# B&R Automation Studio project dbserv_0640 (part 2)

### dbvist.h
```c
/************************************************************************/
/*	Headerfile für DbVist												*/
/*																		*/
/************************************************************************/
#include "pwi_lib.h"

/* Tasknamen für Versionsanzeige */
#define	TASK_DBSERV		"dbserv"
#define	TASK_DBSTCP		"dbstcp"
#define	TASK_DBVIST		"dbvist"
#define	TASK_IEC103		"iec103"
#define	TASK_L2DP		"l2dp"
#define	TASK_IODRV		"iodrv"
#define	TASK_GPS		"gps"

#define	MAX_ITEM			4000	/* max.Anzahl von Items */
#define ANZ_SCAN_AL			64		/* gescannte Alarme pro Zyklus */

#define	MENU_MAIN	1
#define	MENU_ITEM	2
#define	MENU_ALISTE	3
#define	MENU_NODP	5
#define	MENU_SYS	6
#define	MENU_CLOCK	7
#define	MENU_VERSION	8
#define MENU_MAX	10

#define KEY_OPT		33
#define KEY_F		34
#define KEY_STERN	35
#define KEY_ALISTE	39
#define KEY_AP		40
#define KEY_BP		41
#define KEY_AL		42
#define KEY_ZL		43
#define KEY_Q		48
#define KEY_SYS		51
#define KEY_PAGEUP	53
#define KEY_ONEUP	54
#define KEY_PLUS	55
#define KEY_PAGEDWN	56
#define KEY_ONEDWN	57
#define KEY_MINUS	58
#define KEY_UP		59
#define KEY_RIGHT	60
#define KEY_DOWN	61
#define KEY_LEFT	62
#define KEY_HOME	63
#define KEY_ENTER	65

typedef struct {
	STRING	time[32];
} ALTIME_typ;

/*
typedef struct {
	UINT	LifeCheck;
	UINT	TimeOut;
	INT		DefcurNo;
	INT		DefcmdNo;
	INT		NewcurNo;
	INT		NewcmdNo;
	USINT	DefownPage;
	USINT	NewownPage;
	SINT	DefcurPage;
	SINT	NewcurPage;
	USINT	triggerCur;
	USINT	disCursor;
	USINT	disCurLFRG;
	SINT	nextInpENo;
	SINT	nextInpESt;
	USINT	loopInput;
	USINT	disInput;
	USINT	disKey;
	USINT	signKey;
	USINT	dpChar;
	USINT	dpFix;
	USINT	hiddenChar;
	USINT	strInsert;
	USINT	srcKeyLim;
	USINT	curChar;
	USINT	curInput;
	SINT	curPosObj;
	USINT	signFormat;
	USINT	optNewPage;
	USINT	nNCnewPage;
	USINT	nNXnewPage;
	USINT	notValidChar;
} PWI_env;
*/
typedef struct {
	UINT	PwiStep;
	BOOL	okPWI;
	UDINT	idPWI;
	UINT	codePWI;
	UINT	infoPWINo;
	UINT	infoPWILn;
	UINT	waitCycles;
	UINT	stateOut;
	USINT	szTrends[256];
	USINT	SpeechEnab[256];
	UINT	SpeechAct;
	UINT	PageAct;
	BOOL	PageAgain;
	BOOL	PageReady;
	UINT	PageNew;
	UINT	SpeechNew;
	INT		ActcurNo;
	INT		ActcmdNo;
	INT		ActownPage;
	USINT	KeyFieldT[16];
	USINT	KeyField[16];
	USINT	KeyFieldP[16];
	USINT	KeyFieldO[16];
	BOOL	TableauOK;
	BOOL	keypress;
	BOOL	keypuls;
	USINT	keyold;
	USINT	keycode;
	USINT	keycodeTab;
	USINT	messageTab;
	BOOL	enterpuls;
	UINT	stateCanTX;
	UINT	stateCanRX;
	UDINT	idCAN;
	UINT	nodeCAN;
	UINT	errCAN;
	USINT	Device[32];
	UINT	stateRsTX;
	UINT	stateRsRX;
	UDINT	idRS;
	UINT	argc;
	UDINT	argv[32];
	USINT	keyuser;
	USINT	ASCIIuser;
	BOOL	changePuls;
	BOOL	changepuls;
	BOOL	inputopen;
	BOOL	funcInp;
	USINT	funcEnter;
	BOOL	funcInpRun;
	UINT	stateInp;

	UINT	codePwi;
	UINT	infoPwi1;
	UINT	infoPwi2;

	UINT	codeText;
	UINT	infoTextNo;
	UINT	infoTextLn;

	UINT	codeMask;
	UINT	infoMaskNo;
	UINT	infoMaskLn;

	UINT	codePage;
	UINT	infoPageNo;
	UINT	infoPageLn;

	UINT	codeObj;
	UINT	infoObjNo;
	UINT	infoObjLn;

	UINT	codeGrph;
	UINT	infoGrphNo;
	UINT	infoGrphLn;

	UINT	codeTrend;
	UINT	infoTrendNo;
	UINT	infoTrendLn;

	UINT	codeCan;
	UDINT	infoCan1;
	UDINT	infoCan2;

	UINT	codeRs;
	UDINT	infoRs1;
	UDINT	infoRs2;

	PWI_env	envPWI;
} PWI_INTERFACE;

typedef struct {
	STRING	vers_dbserv[40];
	STRING	vers_dbvist[40];
	STRING	vers_dbstcp[40];
	STRING	vers_iec103[40];
	STRING	vers_l2dp[40];
	STRING	vers_iodrv[40];
	STRING	vers_gps[40];
} VERSION_typ;

/*_GLOBAL	UINT	PageAct,PageNew,,SpeechAct,SpeechNew;
_GLOBAL	BOOL	keypuls,;
_GLOBAL	USINT	keycode;
*/
_LOCAL	PWI_INTERFACE	*pPWI_INTERFACE;
_LOCAL	UDINT	lenPWI_INTERFACE;
_LOCAL	UINT	PageLast;
_LOCAL	BOOL	keypuls_old;

_LOCAL	STRING	UstName[32],Filter[32],FilterUnten[41];
_LOCAL	USINT	enableItem[MAX_ITEM];
_LOCAL	INT		UstNr;

_LOCAL	UINT	testUINT;
_LOCAL	UINT	GrpIdx,DTypIdx,DPIdx;
_LOCAL	USINT	enableGrp,enableDT,enableDP,enableOGrp,enableODT,enableODP;
_LOCAL	USINT	enableGrp_old,enableDT_old,indexGrp_old,indexDT_old;
_LOCAL	BOOL	activGrp,activDT,activDP;
_LOCAL	BOOL	activGrp_old,activDT_old;
_LOCAL	BOOL	setClock,enableSet,activSet,setClockStarted;
_LOCAL	RTCtime_typ	RTCtime,RTCtimeSet;
_LOCAL	INT		indexSYS, indexGrp,indexDT,indexDP,indexItem,indexAP,indexBP,indexAL,indexZL,indexALL;
_LOCAL	USINT	minute_old;
_LOCAL	UINT	AnzDPfiltered,LastFiltered;

_LOCAL void (*pInitPic[MENU_MAX])();
_LOCAL void (*pCyclPic[MENU_MAX])();
_LOCAL void (*pKeysPic[MENU_MAX])();

_LOCAL	UDINT	myidBrServer;
_LOCAL	UINT	statePV_xgetadr,CheckPWIerrors	_VAR_RETAIN;
_LOCAL 	UINT	idstat,brstate;
_LOCAL	UINT	scanAL,countAL,aktiveAlarme,countALGRP[MAX_GRP],aktiveAlarmeGrp[MAX_GRP];
_LOCAL	BOOL	SammStoer,GrpStoer[MAX_GRP];
_LOCAL	USINT	LED_Aliste;
_LOCAL	USINT	*pData_extern, *pData_iextern, *pData_intern, *pData_valid, *pData_time, *pData_itime, *pData_writelink, *pData_ieventlink, *pData_ihyst, *pData_ievent;
_LOCAL	UDINT 	length_extern, length_intern, length_iextern, length_valid, length_time, length_itime, length_writelink, length_ieventlink, length_ihyst, length_ievent;
_LOCAL	UINT	infoerror,LatchStatusSetValueItem;
_LOCAL	BOOL	Quitt;
_LOCAL	UINT	quitIndex;
_LOCAL	VERSION_typ	Version;
_LOCAL MoVerStruc_typ MO_ver_struct;
_LOCAL	STRING	TestText1[256],TestText2[256];
_LOCAL	UINT	TestTextNr;
```

### dbv_parse.h
```c
/******************************************************************************
*  Projekt:  DbVist Visualisierung für DbServ
*  Teil:     Parserfunktionen
*  Datei:    dbv_parse.c
*------------------------------------------------------------------------------
*  Revision: 01.00
*  Datum:    04-0-2006
*  Autor:    WAI
*------------------------------------------------------------------------------
*  Funktion:
*------------------------------------------------------------------------------
*  Rev.  | Datum    | Name | Kommentar
*  ------+----------+------+---------------------------------------------------
*  01.00 | 04-06-06 | WAI  | Datei-Erstellung
*        |          |      |
******************************************************************************/
/***********************************************************************/
/* Konstantendefinition                                                */
/***********************************************************************/
#define ERR_MSG_PRE_STRG				"dbv"
#define MAX_ERROR_MSG_LOG				20				/* Anzahl Fehler, die in das Log-Buch eingetragen werden */
/* Bezeichnung der Datenmodule */
#define DATA_OBJEKT_DPLIST		"dplist"
#define DATA_OBJEKT_TYPLIST		"typlist"
#define DATA_OBJEKT_DBVTEXT 	"dbv_text"
#define DATA_OBJEKT_TEXT1 		"text_1"
#define DATA_OBJEKT_TEXT2 		"text_2"
#define DATA_OBJEKT_PAGE 		"page_1"
#define DATA_OBJEKT_OBJ1 		"obj_1"
#define DATA_OBJEKT_OBJ2 		"obj_2"
#define DATA_OBJEKT_OBJ3 		"obj_3"
#define DATA_OBJEKT_OBJ4 		"obj_4"
#define DATA_OBJEKT_OBJ5 		"obj_5"

/* Delimiter */
#define DELIM_ALLGEMEIN_ANF		"<Allgemein>"
#define DELIM_ALLGEMEIN_END		"</Allgemein>"
#define DELIM_DTYP_ANF			"<Dtyp>"
#define DELIM_DTYP_END			"</Dtyp>"
#define DELIM_OBJGRPDTYP_ANF	"<ObjGrpDtyp>"
#define DELIM_OBJGRPDTYP_END	"</ObjGrpDtyp>"
#define DELIM_OBJITEMAP_ANF		"<ObjItemAP>"
#define DELIM_OBJITEMAP_END		"</ObjItemAP>"
#define DELIM_OBJITEMBPAL_ANF	"<ObjItemBPAL>"
#define DELIM_OBJITEMBPAL_END	"</ObjItemBPAL>"
#define DELIM_OBJITEMZL_ANF		"<ObjItemZL>"
#define DELIM_OBJITEMZL_END		"</ObjItemZL>"
#define DELIM_OBJITEMALIST_ANF	"<ObjItemAList>"
#define DELIM_OBJITEMALIST_END	"</ObjItemAList>"
#define DELIM_OBJSYS_ANF		"<ObjSys>"
#define DELIM_OBJSYS_END		"</ObjSys>"
#define DELIM_PAGE_ANF 			"<Page>"
#define DELIM_PAGE_END 			"</Page>"

/* Skalierungsparameter */
#define	MAX_DT					10		/* max.Anzahl von Datentypen */
#define	MAX_GRP					100		/* max.Anzahl von Gruppen */
#define	MAX_UNIT				32		/* max.Anzahl von Einheiten */
#define	MAX_TEXTLIST			32		/* max.Anzahl von Textlisten */
#define	MAX_TEXTVALUE			16		/* max.Wert einer Textliste */

#define BOOL_TYP						"_BOOL"
#define BOOL_IDX						0
#define USINT_TYP						"_USINT"
#define USINT_IDX						1
#define SINT_TYP						"_SINT"
#define SINT_IDX						2
#define UINT_TYP						"_UINT"
#define UINT_IDX						3
#define INT_TYP							"_INT"
#define INT_IDX							4
#define UDINT_TYP						"_UDINT"
#define UDINT_IDX						5
#define DINT_TYP						"_DINT"
#define DINT_IDX						6
#define REAL_TYP						"_REAL"
#define REAL_IDX						8
#define DOUBLE_TYP						"_DOUBLE"
#define DOUBLE_IDX						9

#define DTYP_AP							1
#define DTYP_BP							2
#define DTYP_AL							3
#define DTYP_ZL							4

/*-------------------------------------------------------
	Fehlermeldungen
---------------------------------------------------------*/
#define NO_ERROR						0

/* Fehlermeldungen: Datenmodul nicht gefunden */
#define PARS_ERR_DPLIST_NOT_FOUND		501				/* Fehler: Datenmodul dplist nicht gefunden */
#define PARS_TXT_DPLIST_NOT_FOUND		"datamodule dplist not found"

#define PARS_ERR_TYPLIST_NOT_FOUND		502				/* Fehler: Datenmodul typlist nicht gefunden */
#define PARS_TXT_TYPLIST_NOT_FOUND		"datamodule typlist not found"

#define PARS_ERR_DBVTEXT_NOT_FOUND		503				/* Fehler: Datenmodul dbv_text nicht gefunden */
#define PARS_TXT_DBVTEXT_NOT_FOUND		"datamodule dbv_text not found"

#define PARS_ERR_MEM_ALLOC				504				/* Fehler: Speicher kann nicht allokiert werden */
#define PARS_TXT_MEM_ALLOC				"TMP_alloc not successfull"

#define PARS_ERR_CREATE_DM				505				/* Fehler: Datenmodul kann nicht erzeugt werden */
#define PARS_TXT_CREATE_DM				"Create DM not successfull"

/* Fehlermeldungen des globalen Teiles */
#define PARS_ERR_UNKNOWN_GLOBAL_ENTRY	505				/* Fehler: Unbekannter Eintrag in globalen Bereich */
#define PARS_ERR_GRP_UNKNOWN			506				/* Fehler: Name kann keiner Gruppe zugeordnet werden */
#define PARS_ERR_TO_MUCH_GRP			507				/* Fehler: Anzahl deklarierter Gruppen zu gross  */
#define PARS_ERR_UNIT_UNKNOWN			508				/* Fehler: Name kann keiner Einheit zugeordnet werden */
#define PARS_ERR_TO_MUCH_UNITS			509				/* Fehler: Anzahl deklarierter Einheiten zu gross  */
#define PARS_ERR_TLIST_UNKNOWN			510				/* Fehler: Name kann keiner Textliste zugeordnet werden */
#define PARS_ERR_TO_MUCH_TLISTS			511				/* Fehler: Anzahl deklarierter Textlisten zu gross  */

#define PARS_ERR_DPTYP_NR_NOT_DEFINED	609				/* Fehler: Datentyp Nummer nicht definiert */
#define PARS_ERR_ITEM_NR_NOT_DEFINED	610				/* Fehler: Item Nummer nicht definiert */
#define PARS_ERR_ITEM_TYP_NOT_DEFINED	611				/* Fehler: Item Typ nicht definiert */
#define PARS_ERR_ITEM_TYP_UNKNOWN		612				/* Fehler: Item Typ unbekannt */
#define PARS_ERR_ITEM_NAME_NOT_DEFINED	613				/* Fehler: Item Name nicht definiert */

/* Fehlermeldungen des Itembereiches */
#define PARS_ERR_UNKNOWN_ITEM_ENTRY		700				/* Fehler: Unbekannter Eintrag in Item Bereich (DM typlist)*/
#define PARS_ERR_GRP_NOTDEFINED			701				/* Fehler: Gruppe ist nicht definiert */
#define PARS_ERR_TLIST_NOTDEFINED		702				/* Fehler: Textliste ist nicht definiert */
#define PARS_ERR_ITEM_DTYP_NOT_DEFINED	703				/* Fehler: Datentyp ist nicht definiert */

#define PARS_ERR_REPLACE				710				/* Fehler beim ersetzen von Token */

#define PARS_ERR_PWI_NOT_FOUND			800				/* Fehler: Interface zu PWI nicht gefunden */
#define PARS_ERR_PWI_ERROR				801				/* Fehler: PWI meldet Fehler */
/*-------------------------------------------------------
	Schlüsselworte
---------------------------------------------------------*/
/* Hilfskonstanten */

#define ALL_SECTION						0				/* Es wird im allgemeinen Teil geparst (Meldungsunterdrückung) */
#define DBV_SECTION						1				/* Es wird im VIS - Teil geparst (Meldung bei unbekannten Schlüsselworten) */
#define DP_PART							0				/* Es wird im allgemeinen Datenpunktbereich geparst */
#define ITEM_PART						1				/* Es wird im allgemeinen Itembereich geparst */

/* Schluesselworte Sectionen */
#define	KW_DBV_SECTION					"VIS"			/* Schlüsselwort für VIS-Section */
#define	KW_ALL_SECTION					"ALL"			/* Schlüsselwort für Allgemeine-Section */
#define KW_ITEM_SECTION					"ITEM"			/* Schlüsselwort für ITEM-Section */
#define KW_BLOCK_SECTION				"BLOCK"			/* Schlüsswlwort für Blockdefinition */

/* Schluesselworte  globaler Teil */
#define KW_UST							"UST"			/* Schlüsselwort für UST */
#define KW_VIS_USTNR					"NR"			/* Schlüsselwort für UST-Nummer */
#define KW_VIS_USTNAME					"NAME"			/* Schlüsselwort für UST-Name */
#define KW_VIS_USTIF					"IF"			/* Schlüsselwort für Interface */
#define KW_VIS_GRP						"GRP"			/* Schlüsselwort für Gruppe */
#define KW_VIS_GRPNAME					"NAME"			/* Schlüsselwort für Gruppennamen */
#define KW_VIS_UNIT						"EINH"			/* Schlüsselwort für Einheit */
#define KW_VIS_TLIST					"TLIST"			/* Schlüsselwort für Textliste */
#define KW_VIS_TLISTT0					"T0"			/* Schlüsselwort für Textliste Zusatnd 0*/
#define KW_VIS_TLISTT1					"T1"			/* Schlüsselwort für Textliste Zusatnd 1*/
#define KW_VIS_TLISTT2					"T2"			/* Schlüsselwort für Textliste Zusatnd 2*/
#define KW_VIS_TLISTT3					"T3"			/* Schlüsselwort für Textliste Zusatnd 3*/
#define KW_VIS_TLISTT4					"T4"			/* Schlüsselwort für Textliste Zusatnd 4*/
#define KW_VIS_TLISTT5					"T5"			/* Schlüsselwort für Textliste Zusatnd 5*/
#define KW_VIS_TLISTT6					"T6"			/* Schlüsselwort für Textliste Zusatnd 6*/
#define KW_VIS_TLISTT7					"T7"			/* Schlüsselwort für Textliste Zusatnd 7*/
#define KW_VIS_TLISTT8					"T8"			/* Schlüsselwort für Textliste Zusatnd 8*/
#define KW_VIS_TLISTT9					"T9"			/* Schlüsselwort für Textliste Zusatnd 9*/
#define KW_VIS_TLISTT10					"T10"			/* Schlüsselwort für Textliste Zusatnd 10*/
#define KW_VIS_TLISTT11					"T11"			/* Schlüsselwort für Textliste Zusatnd 11*/
#define KW_VIS_TLISTT12					"T12"			/* Schlüsselwort für Textliste Zusatnd 12*/
#define KW_VIS_TLISTT13					"T13"			/* Schlüsselwort für Textliste Zusatnd 13*/
#define KW_VIS_TLISTT14					"T14"			/* Schlüsselwort für Textliste Zusatnd 14*/
#define KW_VIS_TLISTT15					"T15"			/* Schlüsselwort für Textliste Zusatnd 15*/

/* Schluesselworte  Datenpunkt Teil */
#define KW_DP_ALL_ANL					"ANLAGE"		/* Schlüsselwort für Anlagennummer */
#define KW_DP_ALL_ANL_NR				"NR"			/* Schlüsselwort für Anlagennummer (ANLAGEN.NR) */
#define KW_DP_ALL_DP					"DP"			/* Schlüsselwort für Datenpunktnummer */
#define KW_DP_ALL_DP_NR					"NR"			/* Schlüsselwort für Datenpunktnummer (DP.NR) */
#define KW_DP_ALL_TYP					"TYP"			/* Schlüsselwort für Datenpunkttyp */
#define KW_DP_ALL_ITEM					"ITEM"			/* Schlüsselwort Item Datentyp */
#define KW_DP_ALL_ITEM_TYP				"TYP"			/* Schlüsselwort Item-Datentyp ITEM.TYP */
#define KW_DP_ALL_ITEM_NR				"NR"			/* Schlüsselwort Item-Nummer (ITEM.NR) */

/* Schlüsselworte TYPLIST	ALL-Teil Datenpunkt */
#define	KW_DPTYP_ALL_TYP				"TYP"			/* Schlüsselwort Datentyp Nummer */
#define KW_DPTYP_ALL_TYP_NR				"NR"			/* Schlüsselwort Datentyp Nummer (TYP.NR) */

/* Schlüsselworte TYPLIST	ALL-Teil ITEM */
#define KW_ITEM_ALL_ITEM_TYP			"TYP"			/* Schlüsselwort Item Datentyp */
#define KW_ITEM_ALL_ITEM				"ITEM"			/* Schlüsselwort Item-Nummer */
#define KW_ITEM_ALL_ITEM_NR				"NR"			/* Schlüsselwort Item-Nummer (ITEM.NR) */
#define KW_ITEM_ALL_ITEM_NAME			"NAME"			/* Schlüsselwort Item-Nummer (ITEM.NAME) */
#define KW_ITEM_ALL_ITEM_TEXT			"TEXT"			/* Schlüsselwort Item-Nummer (ITEM.TEXT) */

/* Schlüsselworte TYPLIST	VIS-Teil */
#define KW_ITEM_VIS_GRP					"GRP"			/* Schlüsselwort Gruppe */
#define KW_ITEM_VIS_DTYP				"DTYP"			/* Schlüsselwort Datentyp */
#define KW_ITEM_VIS_EINH				"EINH"			/* Schlüsselwort Einheit */
#define KW_ITEM_VIS_KPOS				"KPOS"			/* Schlüsselwort Kommaposition */
#define KW_ITEM_VIS_TLIST				"TLIST"			/* Schlüsselwort Textliste */
#define KW_ITEM_VIS_QUITT				"QUITT"			/* Schlüsselwort Quittierung */

/* Infos des Parsers */
typedef struct
{
	long					memAdr;
	long					memSize;
	unsigned short			allocStatus;
	plcbit					ErrorMsg;
	unsigned short			NrOfLogEntrys;
	unsigned short			error;
	unsigned short			warning;
	UDINT					OffsPage;
	UDINT					LenPage;
	UDINT					OffsObjGrpDtyp;
	UDINT					LenObjGrpDtyp;
	UDINT					OffsObjItemAP;
	UDINT					LenObjItemAP;
	UDINT					OffsObjItemBPAL;
	UDINT					LenObjItemBPAL;
	UDINT					OffsObjItemZL;
	UDINT					LenObjItemZL;
	UDINT					OffsObjAlist;
	UDINT					LenObjAlist;
	UDINT					OffsObjSys;
	UDINT					LenObjSys;
	UDINT					OffsAllgemein;
	UDINT					LenAllgemein;
	UINT					AnzahlAllgemein;
	UDINT					OffsDtyp;
	UDINT					LenDtyp;
	UINT					AnzahlDtyp;
	unsigned short			NrOfGrp;
	unsigned short			GrpIdx;
	long					GrpNrAct;
	plcbit					GrpNrValid;
	unsigned short			NrOfUnits;
	unsigned short			NrOfTlist;
	unsigned short			TlistIdx;
	long					TlistNrAct;
	plcbit					TlistNrValid;
	unsigned short			NrOfDataPoints;
	unsigned short			NrOfItems;
	unsigned short			NrOfAL;
	unsigned char			*DPName;
	unsigned short			LenDPName;
	unsigned char			*OptName;
	unsigned short			LenOptName;
	unsigned short			LenItemName;
	unsigned short			LenItemText;
	unsigned long			LenAllItemName;
	unsigned long			LenAllItemText;
	unsigned long			LenText1,LenText2;
	long					memAdrText1,memAdrText2,memAdrPage,memAdrObj1,memAdrObj2,memAdrObj3,memAdrObj4,memAdrObj5;
	long					memSizeText1,memSizeText2;
	unsigned short			allocStatusText1,allocStatusText2,allocStatusPage,allocStatusObj1,allocStatusObj2,allocStatusObj3,allocStatusObj4,allocStatusObj5;
	unsigned short			OffsetAllgemein;
	unsigned short			OffsetDtyp;
	unsigned short			OffsetGrp;
	unsigned short			OffsetTextlist;
	unsigned short			OffsetUnit;
	unsigned short			OffsetItems;
	unsigned short			ActItemIdx;
} DBV_ParserInfo_typ;

/* Hilfsvariable des Parsers */
typedef struct {
	unsigned char			*pParser;
	unsigned char			*pParserLine;
	unsigned char			*pParserErr;
	unsigned char			*pDataArg1;
	unsigned char			*pDataArg2;
	unsigned char			*pDataArg3;
	unsigned short			SizeArg1;
	unsigned short			SizeArg2;
	unsigned short			SizeArg3;
	unsigned short			SectionType;
	unsigned short			CountLines;
} Parser_typ;

typedef struct
{
	plcbit					defined;
	unsigned char			*name;
	unsigned short			size;
} DBV_ParserTypInfo_typ;

typedef struct
{
	plcbit					defined;
	long					value;
} DBV_ParserParInfo_typ;

typedef struct
{
	plcbit					defined;
	long					value;
	unsigned char			*name[MAX_TEXTVALUE];
	unsigned short			size[MAX_TEXTVALUE];
} DBV_ParserTlistInfo_typ;

typedef struct
{
	DBV_ParserParInfo_typ	GrpNr;
	DBV_ParserTypInfo_typ	GrpName;
} DBV_ParserGrpInfo_typ;

/* --------------------------*/
/* Globale Parameter         */
/* --------------------------*/

typedef struct
{
	DBV_ParserParInfo_typ	UstNr;
	DBV_ParserTypInfo_typ	UstName;
	DBV_ParserTypInfo_typ	Interface;
	DBV_ParserTypInfo_typ	Dtyp[MAX_DT];
	DBV_ParserGrpInfo_typ	Grp[MAX_GRP];
	DBV_ParserTypInfo_typ	Unit[MAX_UNIT];
	DBV_ParserTlistInfo_typ	Textlist[MAX_TEXTLIST];
} DBV_GlobalData_typ;
/* ----------------------------*/
/* Parameter Datenpunkt / Item */
/* ----------------------------*/

typedef struct
{
	DBV_ParserParInfo_typ	AnlagenNr;
	DBV_ParserParInfo_typ	DPNr;
	DBV_ParserTypInfo_typ	Typ;
	DBV_ParserParInfo_typ	DPTypNr;
	DBV_ParserParInfo_typ	ItemNr;
	DBV_ParserTypInfo_typ	ItemTyp;
	DBV_ParserParInfo_typ	ItemTypNr;
	DBV_ParserTypInfo_typ	ItemName;
	DBV_ParserTypInfo_typ	ItemText;
	DBV_ParserParInfo_typ	GrpNr;
	DBV_ParserParInfo_typ	Dtyp;
	DBV_ParserParInfo_typ	Unit;
	DBV_ParserParInfo_typ	Tlist;
	DBV_ParserParInfo_typ	Kpos;
	DBV_ParserParInfo_typ	Quitt;
	USINT					noVIS;
} DBV_ItemData_typ;

/* Struktur eines Datenpunkt Items im Speicher */
typedef struct {
	UINT	AnlagenNr;						/* Anlagennummer */
	UINT	Device;							/* Devicenummer (immer 1)*/
	UINT	DPTypNr;						/* Datentypnummer */
	UINT	DPNr;							/* Datenpunktnummer */
	UINT	ItemNr;							/* Item Nummer */
	UINT	TextNr;							/* Textnummer im Textpool */
	USINT	GrpNr;							/* Gruppennummer */
	USINT	Dtyp;							/* Datentyp */
	UINT	Unit;							/* Textnummer Einheit im Textpool */
	USINT	Kpos;							/* Komaposition */
	USINT	Tlist;							/* textlist-Nummer */
	USINT	Quitt;							/* Quittier-Datenpunkt */
} DBV_DP_Info_typ;

typedef struct {
	plcbit					showData;
	plcbit					DataValid;
	unsigned short			AnlagenNr;
	unsigned short			DPTypNr;
	unsigned short			DPNr;
	unsigned short			ItemNr;
	DBV_DP_Info_typ 		*pItemData;
	unsigned short			ItemIdx;
} DBV_ItemDiagnose_typ;

/***********************************************************************/
/* Prototypen		                                                   */
/***********************************************************************/
void dbv_parser();
void dbv_parser_err(unsigned short errorNr, unsigned char *pTxtInfo, unsigned char *pTxt0, unsigned char *pTxt1, long info1, unsigned char *pTxt2, long info2, unsigned char *pTxt3, long info3);
void dbv_parser_warn(unsigned short warnNr, unsigned char *pTxtInfo, unsigned char *pTxt0, unsigned char *pTxt1, long info1, unsigned char *pTxt2, long info2, unsigned char *pTxt3, long info3);
int  dbv_parser_sect(USINT *pData, UDINT len, USINT *delim_anf, USINT *delim_end, UDINT *pOffset,UDINT *pLen, UINT *pAnzahl);
void dbv_parser_global();
unsigned char IsANumber(unsigned char *pData);
void dbv_parser_dplist_clear();
void dbv_parser_typlist_clear();
void copyItemData(DBV_ItemData_typ *pItemDest, DBV_ItemData_typ *pItemSrc);
plcbit dbv_parser_iteminfo();
void dbv_parser_dpinfo(plcbit *pBlockFound, plcbit *pDPFound);
plcbit dbv_parser_dptype(unsigned char *pName, unsigned short size);
void dbv_parser_data(unsigned char *pSrcStart,unsigned char *pSrcEnd, Parser_typ *pPa, DBV_ItemData_typ *pData, unsigned char SectionInfo, unsigned char PartInfo);
plcbit dbv_parser_iteminfo_ok(DBV_ItemData_typ *pData);
unsigned char *dbv_findToken(USINT *pSrc,UDINT len,USINT *token);
void dbv_replace_refpab(USINT *pFound,DBV_DP_Info_typ *pDBV_DP_Info);
void dbv_replace_index(USINT *pFound,INT i);
void make_page();
void make_obj1();
void make_obj2();
void make_obj3();
void make_obj4();
void make_obj5();
void get_idBrServer();
void dbv_mem_diagnose();

/**********************************************************
*				Lokale Variablen Declaration
**********************************************************/
_LOCAL	Parser_typ				PaDPList,PaDPListSave;
_LOCAL	Parser_typ				PaTypList,PaTypListSave;

_LOCAL	DatObjInfo_typ			DOI_dplist,DOI_typlist,DOI_dbvtext,DOI_text1,DOI_text2,DOI_page,DOI_obj1,DOI_obj2,DOI_obj3,DOI_obj4,DOI_obj5;
_LOCAL	DatObjDelete_typ		DOD_text1,DOD_text2,DOD_page,DOD_obj1,DOD_obj2,DOD_obj3,DOD_obj4,DOD_obj5;
_LOCAL	DatObjCreate_typ		DOC_text1,DOC_text2,DOC_page,DOC_obj1,DOC_obj2,DOC_obj3,DOC_obj4,DOC_obj5;
_LOCAL	DBV_ParserInfo_typ		DBV_ParserInfo;
_LOCAL	DBV_GlobalData_typ		DBV_GlobalData;
_LOCAL	DBV_ItemData_typ		DBV_DPData,DBV_ItemData,DBV_BlockData;
_LOCAL	signed short			State_find_StationTypPoint, State_find_Section, State_find_Data	_VAR_RETAIN;
_LOCAL	unsigned char			MsgTxt[256];
_LOCAL	UDINT					check_len1,check_len2;

#define ITEM_DIAGNOSE_SIZE		2
_LOCAL	DBV_ItemDiagnose_typ	DBV_ItemDiagnose[ITEM_DIAGNOSE_SIZE];
_LOCAL	DBV_DP_Info_typ 		*pItemData0Diagnose;
_LOCAL	DBV_DP_Info_typ 		*pItemData1Diagnose;

/* Test */
_LOCAL	BOOL					go	_VAR_RETAIN;
```

### eventaprol.h
```c
typedef struct {
	unsigned short	Auftragscode;
	unsigned short	Anlage;
	unsigned short	Unterstation;
	unsigned short	Datentyp;
	unsigned short	Datenpunkt;
	unsigned short	Offset;
	unsigned short	Anzahl;
	unsigned short	res;
	unsigned char	Daten[32];
} EVENT_DOWN;

typedef struct {
	unsigned short	Auftragscode;
	unsigned short	Anlage;
	unsigned short	Unterstation;
	unsigned short	Datentyp;
	unsigned short	Datenpunkt;
	unsigned short	Offset;
	unsigned short	Anzahl;
	unsigned short	res;
} EVENT_DOWN_HEAD;

typedef struct {
	unsigned short	Auftragscode;
	unsigned short	Anlage;
	unsigned short	Unterstation;
	unsigned short	Datentyp;
	unsigned short	Datenpunkt;
	unsigned short	Offset;
	unsigned short	Anzahl;
	unsigned short	res;
	RTCtime_typ		RTCTime;
	unsigned char	Daten[32];
} EVENT_UP;

typedef struct {
	unsigned short	Auftragscode;
	unsigned short	Anlage;
	unsigned short	Unterstation;
	unsigned short	Datentyp;
	unsigned short	Datenpunkt;
	unsigned short	Offset;
	unsigned short	Anzahl;
	unsigned short	res;
	RTCtime_typ		RTCTime;
} EVENT_UP_HEAD;
```

### parser.h
```c
/******************************************************************************
*    COPYRIGHT    BERNECKER + RAINER Industrie-Elektronik Ges.m.b.H           *
*******************************************************************************
*  Projekt:  Burklimat 2000
*  Teil:     Parser-Funktionen
*  Datei:    parser.h
*  Typ:      GNU-C (32 Bit)
*------------------------------------------------------------------------------
*  Revision: 00.25
*  Datum:    26-07-2000
*  Autor:    Martin Kurtz / MKrz
*------------------------------------------------------------------------------
*  Funktion: Globale Include-Datei.
*------------------------------------------------------------------------------
*  Rev.  | Datum    | Name | Kommentar
*  ------+----------+------+---------------------------------------------------
*  00.00 | 23-06-99 | MKrz | Datei-Erstellung
*        |          |      |
******************************************************************************/

/***********************************************************************/
/* Konstantendefinition                                                */
/***********************************************************************/

#define FALSE	0	/* logisch falsch */
#define TRUE	1	/* logisch wahr */

#define cKW_STATION		'&'		/* "&" Stations-Schlüssel */
#define cKW_TYP			'$'		/* "$" Typ-Schlüssel */
#define cKW_ITEM		'§'		/* "/" Item-Schlüssel */
#define cKW_POINT		'@'		/* "@" Punkt-Schlüssel */
#define cKW_OPTION		'~'		/* "~" Options-Schlüssel */
#define cKW_SECTION		'#'		/* "#" Sektions-Schlüssel */

#define cKW_ASSIGNMENT	'='		/* "=" Zuweisungs-Schlüssel */
#define cKW_SEPARATOR	'.'		/* "." Separations-Schlüssel */
#define cKW_STRING		'\''	/* "'" String-Schlüssel */

enum {	cCD_STATION,			/* '&' Stations-Schlüssel */
		cCD_TYP,				/* '$' Typ-Schlüssel */
		cCD_ITEM,				/* '%' Item-Schlüssel */
		cCD_POINT,				/* '@' Punkt-Schlüssel */
		cCD_OPTION,				/* '~' Otions-Schlüssel */
		cCD_SECTION	};			/* '#' Sektions-Schlüssel */

#define cPS_NO_DATA					-1		/* Keine gültigen Daten gefunden */
#define cPS_OPTION_WITHOUT_REF		-2		/* Optioneller Text ohne Station/Typ/Punkt */
#define cPS_NO_REF					-3		/* Station/Typ/Punkt - Bezeichner nicht vorhanden */
#define cPS_KEYWORD_IN_REF			-4		/* Schlüsselwort in Station/Typ/Punkt - Bezeichner */
#define cPS_NO_OPTION				-5		/* Optioneller Text - Bezeichner nicht vorhanden */
#define cPS_KEYWORD_IN_OPTION		-6		/* Schlüsselwort in optionellem Text */
#define cPS_NO_SECTION				-7		/* Sektions - Bezeichner nicht vorhanden */
#define cPS_KEYWORD_IN_SECTION		-8		/* Schlüsselwort in Sektion */
#define cPS_UNEXPECTED_POINT		-9		/* Unerwarteter Punkt */
#define cPS_UNEXPECTED_ASSIGNMENT	-10		/* Unerwartete Zuweisung */

/***********************************************************************/
/* Parser-Funktionen                                                   */
/***********************************************************************/

signed short find_StationTypPoint (unsigned char* pDmStart, unsigned char* pParser, unsigned char* pDmEnd,
									unsigned char** ppParser, unsigned char** ppParserLine,
									unsigned char** ppParserErr, unsigned short* pCountZeroTerms,
									unsigned char** ppDataArg1, unsigned short* pSizeArg1,
									unsigned char** ppDataArg2, unsigned short* pSizeArg2,
									unsigned short* pSectionType );

signed short find_Section (unsigned char* pDmStart, unsigned char* pParser, unsigned char *pDmEnd,
							unsigned char** ppParser, unsigned char** ppParserLine,
							unsigned char** ppParserErr, unsigned short* pCountZeroTerms,
							unsigned char** ppDataArg1, unsigned short* pSizeArg1,
							unsigned char** ppDataArg2, unsigned short* pSizeArg2,
							unsigned char* pSectionName );

signed short find_Data (unsigned char* pDmStart, unsigned char* pParser, unsigned char *pDmEnd,
						 unsigned char** ppParser, unsigned char** ppParserLine,
						 unsigned char** ppParserErr, unsigned short* pCountZeroTerms,
						 unsigned char** ppDataArg1, unsigned short* pSizeArg1,
						 unsigned char** ppDataArg2, unsigned short* pSizeArg2,
						 unsigned char** ppDataArg3, unsigned short* pSizeArg3 );
```

### platform.h
```c
/******************************************************************************
*    COPYRIGHT    BERNECKER + RAINER Industrie-Elektronik Ges.m.b.H           *
*******************************************************************************
*  Projekt:  BrTcp
*  Teil:     Header-File
*  Datei:    platform.h
*  Typ:      GNU C (32 Bit)
*------------------------------------------------------------------------------
*  Revision: 01.00
*  Datum:    04-08-2003
*  Autor:    Martin Kurtz / MKrz
*------------------------------------------------------------------------------
*  Funktion: Generelle Plattform-Definition.
*------------------------------------------------------------------------------
*  Rev.  | Datum    | Name | Kommentar
*  ------+----------+------+---------------------------------------------------
*  01.00 | 04-08-03 | MKrz | Datei-Erstellung
*        | 13-08-03 | RES  | Softwareplattform eingefuegt
*        |          |      |
******************************************************************************/

/* ------------------ */
/* Hardware-Plattform */
/* ------------------ */
#define	INTEL
#undef MOTOROLA

/* ------------------ */
/* Software-Plattform */
/* ------------------ */
#undef BURKLIMAT2000
#define	BRSERVER
```

### Package Logical/DbServ-Basis - DbServ Kernel

### Program Logical/DbServ-Basis/dbserv (ANSIC, version 6.40.0) - DbServ Kernel

- platform.h (reference to Logical/GlobalIncludes/platform.h)

- bksys.h (reference to Logical/GlobalIncludes/bksys.h)

- parser.h (reference to Logical/GlobalIncludes/parser.h)

- dbserv.h (reference to Logical/GlobalIncludes/dbserv.h)

#### parser.c
```c
#ifdef _DEFAULT_INCLUDES
	#include <AsDefault.h>
#endif

/******************************************************************************
*    COPYRIGHT    BERNECKER + RAINER Industrie-Elektronik Ges.m.b.H           *
*******************************************************************************
*  Projekt:  Burklimat 2000
*  Teil:     Parser-Funktionen
*  Datei:    parser.c
*  Typ:      GNU-C (32 Bit)
*------------------------------------------------------------------------------
*  Revision: 00.26
*  Datum:    26-09-2001
*  Autor:    Martin Kurtz / MKrz
*------------------------------------------------------------------------------
*  Funktion: Globale Include-Datei.
*------------------------------------------------------------------------------
*  Rev.  | Datum    | Name | Kommentar
*  ------+----------+------+---------------------------------------------------
*  00.10 | 03-11-99 | MKrz | Datei-Erstellung
*  00.25 | 26-07-00 | MKrz |
*        | 21-09-01 | Res  | burtrap ersetzt durch sys_lib
*  00.26 | 26-09-01 | Res  | #include <dvframe.h> entfernt (wird nicht benoetigt)
*  02.00 | 11-09-06 | Wai  | find_StationTypPoint: Verwendung von if/elseif statt switch
*							 wegen §-Bezeichner
******************************************************************************/

/***********************************************************************/
/* Headerfiles einbinden                                               */
/***********************************************************************/

#include <bur\plc.h>		/* RPS-spezifische Typendeklarationen */
#include <sys_lib.h>		/* 21.09.01/RES: Ersatz fuer <burtrap.h> */

#include <string.h>			/* String-Library */

#include "parser.h"			/* Parser-spezifische Typendeklarationen */

/***********************************************************************/
/* Parser-Funktionen                                                   */
/***********************************************************************/

signed short find_StationTypPoint (unsigned char* pDmStart, unsigned char* pParser, unsigned char* pDmEnd,
									unsigned char** ppParser, unsigned char** ppParserLine,
									unsigned char** ppParserErr, unsigned short* pCountZeroTerms,
									unsigned char** ppDataArg1, unsigned short* pSizeArg1,
									unsigned char** ppDataArg2, unsigned short* pSizeArg2,
									unsigned short* pSectionType )
{
	unsigned char	*pDM;
	unsigned short	ParserState = 0;
	signed short	ParserError = FALSE;

	/* Pointer Arg1..Arg2 initialisieren */
	*ppDataArg1 = NULL;
	*ppDataArg2 = NULL;

	/* Textlängen der Arg1..Arg2 initialisieren */
	*pSizeArg1 = 0;
	*pSizeArg2 = 0;

	/* Line-Pointer initialisieren */
	if (pParser == pDmStart)
		*ppParserLine = pDmStart;
	else {
		*ppParserLine = pParser;
		while (*ppParserLine > pDmStart && !(**ppParserLine != 0 && *(*ppParserLine-1) == 0))
			(*ppParserLine)--;
	}

	/* Parse über Datenmodul */
	for (pDM = pParser; pDM < pDmEnd; pDM++, *ppParser = pDM, *ppParserErr = pDM)
	{
		/* Nullterminierungen des Datenmodules zählen */
		if (pCountZeroTerms != NULL) {
			if (*pDM == 0)
				(*pCountZeroTerms)++;
		}

		/* neuer Line-Pointer ? */
		if (pDM > pParser && *pDM != 0 && *(pDM-1) == 0)
			*ppParserLine = pDM;

		/* DFA */
		switch (ParserState)
		{
			/* Suche nach erstem Schlüsselwort */
			case 0:
				if (*pDM == (unsigned char) cKW_STATION || *pDM == (unsigned char) cKW_TYP ||
					*pDM == (unsigned char) cKW_ITEM || *pDM == (unsigned char) cKW_POINT)
				{
					switch ((char)*pDM)
					{
						case cKW_STATION:
							*pSectionType = cCD_STATION;
							break;

						case cKW_TYP:
							*pSectionType = cCD_TYP;
							break;

						case cKW_ITEM:
							*pSectionType = cCD_ITEM;
							break;

						case cKW_POINT:
							*pSectionType = cCD_POINT;
							break;
					}
					ParserState = 1;
					break;
				}
				else if (*pDM == cKW_OPTION)
				{
					ParserError = cPS_OPTION_WITHOUT_REF;
					ParserState = 5;
					break;
				}
				break;

			/* Suche nach Schlüsselwort - Bezeichner */
			case 1:
				if (*pDM == 0) {
					if (*ppDataArg1 != NULL) {
						ParserState = 2;
						break;
					}
					else {
						ParserError = cPS_NO_REF;
						ParserState = 5;
						break;
					}
					break;
				}
				else if (*pDM == ' ' || *pDM == '\t') {
					break;
				}
				else
				{
					if (*pDM == (unsigned char) cKW_STATION || *pDM == (unsigned char) cKW_TYP ||
						*pDM == (unsigned char) cKW_ITEM || *pDM == (unsigned char) cKW_POINT ||
						*pDM == (unsigned char) cKW_OPTION || *pDM == (unsigned char) cKW_SECTION)
					{
						ParserError = cPS_KEYWORD_IN_REF;
						ParserState = 5;
						break;
					}
					else
					{
						/* Buchstaben eines Schlüsselwort-Bezeichners gefunden */
						if (*ppDataArg1 == NULL)
							*ppDataArg1 = pDM;

						/* Länge des Schlüsselwort-Bezeichners erhöhen */
						if (*ppDataArg1 != NULL)
							(*pSizeArg1)++;
						break;
					}
					break;
				}
				break;

			/* Suche nach optionalem Text */
			case 2:
				if (*pDM == (unsigned char) cKW_OPTION) {
					ParserState = 3;
					break;
				}
				if (*pDM == (unsigned char) cKW_STATION || *pDM == (unsigned char) cKW_TYP ||
					*pDM == (unsigned char) cKW_ITEM || *pDM == (unsigned char) cKW_POINT ||
					*pDM == (unsigned char) cKW_SECTION)
				{
					ParserState = 4;
					break;
				}
				break;

			/* Suche nach optionellem Text - Bezeicher */
			case 3:
				if (*pDM == 0) {
					if (*ppDataArg2 != NULL) {
						ParserState = 4;
						break;
					}
					else {
						*ppDataArg2 = pDM;
						ParserState = 4;

					/*	ParserError = cPS_NO_OPTION;
						ParserState = 5;*/
						break;
					}
					break;
				}
				if (*pDM == (unsigned char) cKW_STATION || *pDM == (unsigned char) cKW_TYP ||
					*pDM == (unsigned char) cKW_ITEM || *pDM == (unsigned char) cKW_POINT ||
					*pDM == (unsigned char) cKW_OPTION || *pDM == (unsigned char) cKW_SECTION)
				{
					ParserError = cPS_KEYWORD_IN_OPTION;
					ParserState = 5;
					break;
				}
				else
				{
					/* Buchstaben eines Schlüsselwort-Bezeichners gefunden */
					if (*ppDataArg2 == NULL)
						*ppDataArg2 = pDM;

						/* Länge des Schlüsselwort-Bezeichners erhöhen */
					if (*ppDataArg2 != NULL)
							(*pSizeArg2)++;
					break;
				}
				break;

			/* Paser korrekt beenden */
			case 4:
				break;

			/* Parser mit Fehlerzustand beenden */
			case 5:
				break;
		} /* (ParserState) */
		if (ParserState == 4 || ParserState == 5)
			break;
	} /* (pDM = pParser; pDM < pDmEnd; pDM++, *ppParser = pDM, *ppParserErr = pDM) */

	/* Nullterminierungen des Datenmodules nur einmal zählen */
	if (**ppParser == 0)
		(*ppParser)++;

	/* Pointer mindestens ein Zeichen weiter stellen */
	if (*ppParser == pParser)
		(*ppParser)++;

	/* DFA_Zustand: Suche nach optionalem Text */
	if (ParserState == 2)
		return TRUE;

	/* DFA_Endzustand ohne Fehler */
	if (ParserState == 4)
		return TRUE;

	/* DFA_Endzustand mit Fehler */
	if (ParserState == 5)
		return ParserError;

	/* DFA ohne Endzustand abgebrochen */
	return cPS_NO_DATA;
}

signed short find_Section (unsigned char* pDmStart, unsigned char* pParser, unsigned char *pDmEnd,
							unsigned char** ppParser, unsigned char** ppParserLine,
							unsigned char** ppParserErr, unsigned short* pCountZeroTerms,
							unsigned char** ppDataArg1, unsigned short* pSizeArg1,
							unsigned char** ppDataArg2, unsigned short* pSizeArg2,
							unsigned char* pSectionName )
{
	unsigned char	*pDM;
	unsigned short	ParserState = 0;
	signed short	ParserError = FALSE;
	unsigned short	i;
	size_t			lenSectionName;

	/* Pointer Arg1..Arg2 initialisieren */
	*ppDataArg1 = NULL;
	*ppDataArg2 = NULL;

	/* Textlängen der Arg1..Arg2 initialisieren */
	*pSizeArg1 = 0;
	*pSizeArg2 = 0;

	/* Line-Pointer initialisieren */
	if (pParser == pDmStart)
		*ppParserLine = pDmStart;
	else {
		*ppParserLine = pParser;
		while (*ppParserLine > pDmStart && !(**ppParserLine != 0 && *(*ppParserLine-1) == 0))
			(*ppParserLine)--;
	}

	/* Parse über Datenmodul */
	for (pDM = pParser; pDM < pDmEnd; pDM++, *ppParser = pDM, *ppParserErr = pDM)
	{
		/* Nullterminierungen des Datenmodules zählen */
		if (pCountZeroTerms != NULL) {
			if (*pDM == 0)
				(*pCountZeroTerms)++;
		}

		/* neuer Line-Pointer ? */
		if (pDM > pParser && *pDM != 0 && *(pDM-1) == 0)
			*ppParserLine = pDM;

		/* DFA */
		switch (ParserState)
		{
			/* Suche nach erstem Schlüsselwort */
			case 0:
				if (*pDM == (unsigned char) cKW_STATION || *pDM == (unsigned char) cKW_TYP ||
					*pDM == (unsigned char) cKW_ITEM || *pDM == (unsigned char) cKW_POINT ||
					*pDM == (unsigned char) cKW_OPTION)
				{
					ParserError = cPS_NO_DATA;
					ParserState = 3;
					break;
				}
				if (*pDM == cKW_SECTION)
				{
					ParserState = 1;
					break;
				}
				break;

			/* Suche nach Schlüsselwort - Bezeichner */
			case 1:
				if (*pDM == 0) {
					if (*ppDataArg1 != NULL) {
						ParserState = 2;
						break;
					}
					else {
						ParserError = cPS_NO_SECTION;
						ParserState = 3;
						break;
					}
					break;
				}
				else if (*pDM == ' ' || *pDM == '\t') {
					break;
				}
				else
				{
					if (*pDM == (unsigned char) cKW_STATION || *pDM == (unsigned char) cKW_TYP ||
						*pDM == (unsigned char) cKW_ITEM || *pDM == (unsigned char) cKW_POINT ||
						*pDM == (unsigned char) cKW_OPTION || *pDM == (unsigned char) cKW_SECTION)
					{
						if (*ppDataArg1 == NULL) {
							ParserError = cPS_KEYWORD_IN_REF;
							ParserState = 3;
							break;
						}
						else {
							ParserState = 2;
							break;
						}
						break;
					}
					else
					{
						if (*ppDataArg1 == NULL) {
							*ppDataArg1 = pDM;
							lenSectionName = strlen (pSectionName);
							for (i = 0; i < lenSectionName; i++) {
								if (*(pDM + i) != *(pSectionName + i)) {
									*ppDataArg1 = NULL;
									break;
								}
							}
							if (*ppDataArg1 != NULL) {
								*pSizeArg1 = lenSectionName;
								*ppDataArg2 = pDM + lenSectionName;
								*pSizeArg2 = lenSectionName;
								break;
							}
							else {
								/* Falsche Sektion */
								ParserState = 0;
								break;
							}
							break;
						}
						if (*ppDataArg1 != NULL) {

							/* Länge des Schlüsselwort-Bezeichners erhöhen */
							if (*ppDataArg2 != NULL && *ppDataArg2 < pDM)
								*pSizeArg2 = pDM - *ppDataArg2 + 1;
							break;
						}
						break;
					}
					break;
				}
				break;

			/* Paser korrekt beenden */
			case 2:
				break;

			/* Parser mit Fehlerzustand beenden */
			case 3:
				break;
		} /* (ParserState) */
		if (ParserState == 2 || ParserState == 3)
			break;
	} /* (pDM = pParser; pDM < pDmEnd; pDM++, *ppParser = pDM, *ppParserErr = pDM) */

	/* Nullterminierungen des Datenmodules nur einmal zählen */
	if (**ppParser == 0)
		(*ppParser)++;

	/* Nullterminierungen des Datenmodules nur einmal zählen */
	if (pCountZeroTerms != NULL) {
		if (*pDM == 0)
			(*pCountZeroTerms)--;
	}

	/* DFA_Endzustand ohne Fehler */
	if (ParserState == 2)
		return TRUE;

	/* DFA_Endzustand mit Fehler */
	if (ParserState == 3)
		return ParserError;

	/* DFA ohne Endzustand abgebrochen */
	return cPS_NO_DATA;
}

signed short find_Data (unsigned char* pDmStart, unsigned char* pParser, unsigned char *pDmEnd,
						 unsigned char** ppParser, unsigned char** ppParserLine,
						 unsigned char** ppParserErr, unsigned short* pCountZeroTerms,
						 unsigned char** ppDataArg1, unsigned short* pSizeArg1,
						 unsigned char** ppDataArg2, unsigned short* pSizeArg2,
						 unsigned char** ppDataArg3, unsigned short* pSizeArg3 )
{
	unsigned char	*pDM;
	unsigned short	ParserState = 0;
	signed short	ParserError = FALSE;

	/* Pointer Arg1..Arg3 initialisieren */
	*ppDataArg1 = NULL;
	*ppDataArg2 = NULL;
	*ppDataArg3 = NULL;

	/* Textlängen der Arg1..Arg3 initialisieren */
	*pSizeArg1 = 0;
	*pSizeArg2 = 0;
	*pSizeArg3 = 0;

	/* Line-Pointer initialisieren */
	if (pParser == pDmStart)
		*ppParserLine = pDmStart;
	else {
		*ppParserLine = pParser;
		while (*ppParserLine > pDmStart && !(**ppParserLine != 0 && *(*ppParserLine-1) == 0))
			(*ppParserLine)--;
	}

	/* Parse über Datenmodul */
	for (pDM = pParser; pDM < pDmEnd; pDM++, *ppParser = pDM, *ppParserErr = pDM)
	{
		/* Nullterminierungen des Datenmodules zählen */
		if (pCountZeroTerms != NULL) {
			if (*pDM == 0)
				(*pCountZeroTerms)++;
		}

		/* neuer Line-Pointer ? */
		if (pDM > pParser && *pDM != 0 && *(pDM-1) == 0)
			*ppParserLine = pDM;

		/* DFA */
		switch (ParserState)
		{
			/* Suche nach erstem Zeichen */
			case 0:
				/* Schlüsselwort gefunden */
				if (*pDM == (unsigned char) cKW_STATION || *pDM == (unsigned char) cKW_TYP ||
					*pDM == (unsigned char) cKW_ITEM || *pDM == (unsigned char) cKW_POINT ||
					*pDM == (unsigned char) cKW_OPTION || *pDM == (unsigned char) cKW_SECTION)
				{
					ParserError = cPS_KEYWORD_IN_SECTION;
					ParserState = 5;
					break;
				}
				else if (*pDM == 0) {
					ParserError = cPS_NO_DATA;
					ParserState = 5;
					break;
				}
				else if (*pDM == ' ' || *pDM == '\t') {
					break;
				}
				else {
					/* Buchstaben eines Argument1 - Bezeichners gefunden */
					if (*ppDataArg1 == NULL)
						*ppDataArg1 = pDM;

					/* Länge des Argument1 - Bezeichners erhöhen */
					if (*ppDataArg1 != NULL)
						(*pSizeArg1)++;

					ParserState = 1;
					break;
				}
				break;

			/* Suche nach pre '.' - Bezeichner */
			case 1:
				if (*pDM == 0) {
					if (*ppDataArg1 != NULL) {
						ParserState = 4;
						break;
					}
					else {
						ParserError = cPS_NO_DATA;
						ParserState = 5;
						break;
					}
					break;
				}
				else if (*pDM == ' ' || *pDM == '\t') {
					if (*ppDataArg1 != NULL) {
						ParserState = 2;
					}
					break;
				}
				else if (*pDM == cKW_SEPARATOR) {
					if (*ppDataArg1 != NULL) {
						ParserState = 2;
						break;
					}
					else {
						ParserError = cPS_NO_DATA;
						ParserState = 5;
						break;
					}
					break;
				}
				else if (*pDM == cKW_ASSIGNMENT) {
					if (*ppDataArg1 != NULL) {
						ParserState = 3;
						break;
					}
					else {
						ParserError = cPS_NO_DATA;
						ParserState = 5;
						break;
					}
					break;
				}
				else
				{
					if (*pDM == (unsigned char) cKW_STATION || *pDM == (unsigned char) cKW_TYP ||
						*pDM == (unsigned char) cKW_ITEM || *pDM == (unsigned char) cKW_POINT ||
						*pDM == (unsigned char) cKW_SECTION || *pDM == (unsigned char) cKW_OPTION)
					{
						ParserError = cPS_KEYWORD_IN_SECTION;
						ParserState = 5;
						break;
					}
					else
					{
						/* Buchstaben eines Argument1 - Bezeichners gefunden */
						if (*ppDataArg1 == NULL)
							*ppDataArg1 = pDM;

						/* Länge des Argument1 - Bezeichners erhöhen */
						if (*ppDataArg1 != NULL)
							(*pSizeArg1)++;
						break;
					}
					break;
				}
				break;

			/* Suche nach post '.' - Bezeichner */
			case 2:
				if (*pDM == 0)
				{
					if (*ppDataArg1 != NULL) {
						ParserState = 4;
						break;
					}
					else {
						ParserError = cPS_NO_DATA;
						ParserState = 5;
						break;
					}
					break;
				}
				else if (*pDM == ' ' || *pDM == '\t') {
					if (*ppDataArg3 != NULL) {
						ParserState = 3;
						break;
					}
				}
				else if (*pDM == cKW_SEPARATOR) {
					ParserError = cPS_UNEXPECTED_POINT;
					ParserState = 5;
					break;
				}
				else if (*pDM == cKW_ASSIGNMENT) {
					ParserState = 3;
					break;
				}
				else
				{
					if (*pDM == (unsigned char) cKW_STATION || *pDM == (unsigned char) cKW_TYP ||
						*pDM == (unsigned char) cKW_ITEM || *pDM == (unsigned char) cKW_POINT ||
						*pDM == (unsigned char) cKW_SECTION || *pDM == (unsigned char) cKW_OPTION)
					{
						ParserError = cPS_KEYWORD_IN_SECTION;
						ParserState = 5;
						break;
					}
					else
					{
						/* Buchstaben eines Argument2 - Bezeichners gefunden */
						if (*ppDataArg2 == NULL)
							*ppDataArg2 = pDM;

						/* Länge des Argument2 - Bezeichners erhöhen */
						if (*ppDataArg2 != NULL)
							(*pSizeArg2)++;
						break;
					}
					break;
				}
				break;

			/* Suche nach post '=' - Bezeichner */
			case 3:
				if (*pDM == 0)
				{
					if (*ppDataArg3 != NULL) {
						ParserState = 4;
						break;
					}
					else {
						ParserError = cPS_NO_DATA;
						ParserState = 5;
						break;
					}
					break;
				}
				else if (*pDM == cKW_STRING)
				{
					ParserState = 6;
					break;
				}
				else if (*pDM == ' ' || *pDM == '\t')
				{
					if (*ppDataArg3 != NULL) {
						ParserState = 4;
					}
					break;
				}
				/*else if (*pDM == cKW_SEPARATOR) {
					ParserError = cPS_UNEXPECTED_POINT;
					ParserState = 5;
					break;
				}*/
				else if (*pDM == cKW_ASSIGNMENT) {
					ParserError = cPS_UNEXPECTED_ASSIGNMENT;
					ParserState = 5;
					break;
				}
				else
				{
					if (*pDM == (unsigned char) cKW_STATION || *pDM == (unsigned char) cKW_TYP ||
						*pDM == (unsigned char) cKW_ITEM || *pDM == (unsigned char) cKW_POINT ||
						*pDM == (unsigned char) cKW_SECTION || *pDM == (unsigned char) cKW_OPTION)
					{
						ParserError = cPS_KEYWORD_IN_SECTION;
						ParserState = 5;
						break;
					}
					else
					{
						/* Buchstaben eines Argument3 - Bezeichners gefunden */
						if (*ppDataArg3 == NULL)
							*ppDataArg3 = pDM;

						/* Länge des Argument3 - Bezeichners erhöhen */
						if (*ppDataArg3 != NULL)
							(*pSizeArg3)++;
						break;
					}
					break;
				}
				break;

			/* Suche nach post ''' - Bezeichner */
			case 6:
				if (*pDM == 0)
				{
					ParserError = cPS_NO_DATA;
					ParserState = 5;
					break;
				}
				else if (*pDM == cKW_STRING)
				{
					if (*ppDataArg3 != NULL) {
						(*ppParser)++;
						ParserState = 4;
						break;
					}
					else {
						ParserError = cPS_NO_DATA;
						ParserState = 5;
						break;
					}
					break;
				}
				else
				{
					/* Buchstaben eines Argument3 - Bezeichners gefunden */
					if (*ppDataArg3 == NULL)
						*ppDataArg3 = pDM;

					/* Länge des Argument3 - Bezeichners erhöhen */
					if (*ppDataArg3 != NULL)
						(*pSizeArg3)++;
					break;
				}
				break;

			/* Paser korrekt beenden */
			case 4:
				break;

			/* Parser mit Fehlerzustand beenden */
			case 5:
				break;
		} /* (ParserState) */
		if (ParserState == 4 || ParserState == 5)
			break;
	} /* (pDM = pParser; pDM < pDmEnd; pDM++, *ppParser = pDM, *ppParserErr = pDM) */

	/* Nullterminierungen des Datenmodules nur einmal zählen */
	if (pCountZeroTerms != NULL) {
		if (*pDM == 0)
			(*pCountZeroTerms)--;
	}

	/* DFA_Endzustand ohne Fehler */
	if (ParserState == 4)
		return TRUE;

	/* DFA_Endzustand mit Fehler */
	if (ParserState == 5)
		return ParserError;

	/* DFA ohne Endzustand abgebrochen */
	return cPS_NO_DATA;
}
```

#### bksysall.c
```c
#ifdef _DEFAULT_INCLUDES
	#include <AsDefault.h>
#endif
/* bksysall.c ----------------------------------------------------------------- */

#include <bur/plc.h>      /*some usefull macros for B&R pcc programming*/
#include <sys_lib.h>

#include <stdlib.h>
#include <string.h>

#include "bksys.h"

/*-----------------------------------------------------------------------------
// ErrStatistics
// Fehlerbehandlungsroutine
// Last Edit:
//		28.06.00/RES:	Bei mehrzeiligen Eintraegen wird ab Zeile 2 die Zeilennummer eingetragen
//		12.05.00/RES:	ErrNum=0 wird nicht mehr statistisch erfasst
//						pErrPre eingefuehrt
//						Aufteilung langer ErrTexte auf mehrere Logbuch-Eintraege
//						wobei bedingte und unbedingte Umbrueche definiert werden koennen
//		23.12.99/RES
//		30.04.99/RES
//
// inputs:	ErrStat		Fehlerstatus: 0=Warn, 1=Err, 2=Err+Log, 3=Err+Log+HALT
//			ErrNum		Fehlernummer
//			ErrInfo		Fehlerinfo
//			pErrPre		Praefix zu Fehlertext (fuer jede Eintragszeile)
//			pErrText	Zeiger auf Fehlertext
//
// outputs:
//
// return:
//---------------------------------------------------------------------------*/
void ErrStatistics( unsigned char *pTaskName,
					unsigned char ErrStat, unsigned short ErrNum, unsigned long ErrInfo,
					unsigned char *pErrPre, unsigned char *pErrText )
{
	static Stats_Typ *pStats = NULL;
	static short ErrFlag = 0;
	unsigned short LogErrNo;
	long lPtr, lVarLen;
	char szText[ERRTEXT_MAXLEN + 1];				/* Puffer fuer Fehlertext */
	char *pRead, *pWrite, *pStart, *pReadTemp;		/* Diverse Textzeiger */
	char buffer[64];
	short sByteAnz, sRest, sTextLen, sLine, sReadyText, sReadyLine, sSearchCount, sSearchCountMax;
	short sCutFlag = 0;		/* Trenn-Flag fuer Anzeige des Trennzeichens am Zeilenanfang */

	LogErrNo = EC_BK2_BASE + ErrNum;	/* Fehlernummer fuer Logbuch und LastErr sowie LastWarn */

	if( pStats == NULL ) {	/* Zeiger noch nicht bekannt ? */
		/* Zeiger auf Statistikstruktur ermitteln */
		if (strlen(pTaskName) > 0) {
			strcpy(buffer, pTaskName);
			strcat(buffer, ":");
		}
		else {
			buffer[0] = 0;
		}
		strcat(buffer, "SYS_Statistic");
		if( !PV_xgetadr( buffer, &lPtr, &lVarLen ) ) {
			pStats = (Stats_Typ *)lPtr;
		}
		else {	/* SYS_Statistic nicht bekannt */
			if( ErrFlag == 0 ) {
				ERRxwarning( EC_BK2_BASE + EC_SYS_BASE + NOVALIDSTATSPTR_NUM, 0, NOVALIDSTATSPTR_TEXT );
				ErrFlag = 1;
			}
		}
	}
	if( pStats != NULL ) {	/* Zeiger bekannt ? */
		switch(ErrStat) {
			case WARN:	/* Warnmeldung */
				if( ErrNum > 0 ) {
					pStats->LastWarn = LogErrNo;
				}
				break;
			case ERR:	/* Fehlermeldung ohne Logbucheintrag */
				if( ErrNum > 0 ) {
					pStats->LastErr = LogErrNo;
				}
				break;
			case ERRLOG:		/* Fehlermeldung mit Logbucheintrag */
			case ERRLOGHALT:	/* Fehlermeldung mit Logbucheintrag und RPS-Halt */
				/* Fehlernummer eintragen */
				if( ErrNum > 0 ) {
					pStats->LastErr = LogErrNo;
				}
				/* Praefix in Textpuffer eintragen */
				sByteAnz = strlen( pErrPre );
				if( sByteAnz > 0 ) {	/* Praefix vorhanden! */
					if( sByteAnz >= ERRTEXT_MAXLEN ) {	/* Praefix laenger als Puffer ? */
						sByteAnz = ERRTEXT_MAXLEN - 1;
					}
					strncpy( szText, pErrPre, sByteAnz );
					pStart = szText + sByteAnz;
				}
				else {	/* Kein Praefix angegeben! */
					pStart = szText;
				}
				sTextLen = ERRTEXT_MAXLEN - ( pStart - szText );

				/* Fehlertext zeilenweise in Textpuffer eintragen und ins Logbuch schreiben */
				for( pRead = pErrText, sLine = 0, sReadyText = 0; !sReadyText && sLine < ERRTEXT_MAXLINES; sLine++ ) {
					pWrite = pStart;
					sRest = sTextLen;
					/* Zeilennummer fuer Folgezeilen einfuegen */
					if( sLine > 0 ) {
						if( sRest > 2 ) {	/* Nur, wenn mehr als 2 Zeichen fuer Nutztext zur Verfuegung! */
							*pWrite++ = '1' + sLine;
							sRest--;
						}
					}
					/* Prefic-Trennzeichen einfuegen */
					if( sRest > 2 ) {	/* Nur, wenn mehr als 2 Zeichen fuer Nutztext zur Verfuegung! */
						*pWrite++ = ':';
						sRest--;
					}

					/* Text fuer eine Meldezeile zusammenstellen */
					for( sReadyLine = 0; !sReadyLine && sRest > 0; sRest-- ) {
						/* Trennzeichen an Zeilenanfang einfuegen, wenn letzte Zeile abgeschnitten wurden */
						if( sCutFlag ) {
							sCutFlag = 0;
							if( sRest > 2 ) {	/* Nur, wenn mehr als 2 Zeichen fuer Nutztext zur Verfuegung! */
								*pWrite++ = CUT_SIGN;
								sRest--;
							}
						}
						/* Naechstes Lesezeichen auswerten */
						switch( *pRead  ) {
							case 0:		/* Ende des Fehlertextes erreicht */
								sReadyText = 1;
								sReadyLine = 1;
								break;
							case '\n':	/* Unbedingter Umbruch */
								sReadyLine = 1;
								pRead++;
								break;
							default:	/* Zu druckendes Textzeichen */
								if( sRest == 1 ) {	/* Zeilenende erreicht */
									switch( *( pRead + 1 ) ) {	/* Nachfolgendes Zeichen pruefen */
										case 0:		/* Ende des Fehlertextes erreicht */
											*pWrite++ = *pRead++;
											break;
										case '\n':	/* Unbedingter Umbruch */
										case '\t':	/* Bedingter Umbruch */
										case ' ':	/* Bedingter Umbruch */
											*pWrite++ = *pRead++;
											pRead++;	/* Trennzeichen ueberspringen */
											break;
										default:	/* Kein Trenn bzw. Endezeichen */
											/* Maximale Zeichenanzahl fuer nachfolgende Trennzeichensuche ermitteln */
											sSearchCountMax = ( SEARCH_COUNT_MAX < sTextLen ) ? SEARCH_COUNT_MAX : sTextLen;
											if( (short)strlen( pRead ) < sSearchCountMax ) {
												sSearchCountMax = strlen( pRead );
											}
											/* Letztes bedingtes Trennzeichen suchen */
											for( pReadTemp = pRead - 1, sSearchCount = 1; sSearchCount < sSearchCountMax; pReadTemp--, sSearchCount++ ) {
												if( *pReadTemp == ' ' || *pReadTemp == '\t' ) {
													break;	/* Trennzeichen gefunden => Suche abbrechen */
												}
											}
											if( sSearchCount < sSearchCountMax ) {	/* Suche vorzeitig abgebrochen, d.h. Trennzeichen gefunden */
												pRead -= sSearchCount - 1;	/* Lesezeiger auf Zeichen nach Trennzeichen setzen */
												pWrite -= sSearchCount;	/* Schreibzeiger auf Trennzeichen zuruecksetzen */
											}
											else {	/* Kein Trennzeichen gefunden => Zeile abschneiden */
												*pWrite++ = CUT_SIGN;	/* Kennzeichen fuer "harte" Trennung einfuegen */
												sCutFlag = 1;	/* Trenn-Flag fuer naechste Zeile merken */
											}
											break;
									} /* switch( *pRead ) */
								} /* if( sRest == 1 ) */
								else {	/* Noch nicht am Zeilenende ! */
									*pWrite++ = *pRead++;
								}
								break;
						} /* switch( *pRead ) */
					} /* Zeichenschleife */
					*pWrite = 0;	/* Zeichenkette abschliessen */

					/* Gesamte Zeile ins Logbuch schreiben */
					ERRxwarning( LogErrNo, bin_to_bcd_8( ErrInfo ), szText );

					/* Sonderfall "Textende gleich nach Zeilenende" pruefen */
					if( !sReadyText && *pRead == 0 ) {
						sReadyText = 1;	/*Textende-Flag setzen, um abschließende Leerzeile zu unterdruecken */
					}
				} /* Zeilenschleife */

				/* RPS anhalten ? */
				if( ErrStat == ERRLOGHALT ) {
					ERR_fatal( LogErrNo, bin_to_bcd_8( ErrInfo ) );
				}
				break;
			default:
				break;
		}
		/* Fehlerzaehler erhoehen */
		if( ErrNum > 0 && ErrNum < ERRCNTANZ ){
			if( pStats->ErrCount[ErrNum] < 65535 ) {
				pStats->ErrCount[ErrNum]++;
			}
		}
	}
}

/*-----------------------------------------------------------------------------
// ErrStatisticsX
// Erweiterte Fehlerbehandlungsroutine
// Variante 1: ErrBit entspricht Bitmuster in Fehlermaske ( 2-Byte )
// Last Edit:
//		10.05.00/RES:	pErrPre eingefuehrt
//		23.12.99/RES
//		19.05.99/RES
//
// inputs:  pErrMk		Zeiger auf Fehlermaske
//			ErrBit		Fehlerbit in Fehlermaske
// 			pSyErr  	Zeiger auf Systemfehlerzaehler
//			ErrStat1	Fehlerstatus 1. Auftreten des Fehlers: 0=Warn, 1=Err, 2=Err+Log, 3=Err+Log+HALT
//			ErrStatN	Fehlerstatus n. Auftreten des Fehlers: 0=Warn, 1=Err, 2=Err+Log, 3=Err+Log+HALT
//			ErrNum		Fehlernummer
//			ErrInfo		Fehlerinfo
//			pErrPre		Praefix zu Fehlertext (fuer jede Eintragszeile)
//			pErrText	Zeiger auf Fehlertext
//
// outputs:
//
// return:
//---------------------------------------------------------------------------*/
void ErrStatisticsX(unsigned char *pTaskName,
					unsigned short *pErrMk, unsigned short ErrBit, unsigned short *pSyErr,
					unsigned char ErrStat1, unsigned char ErrStatN, unsigned short ErrNum,
					unsigned long ErrInfo, unsigned char *pErrPre, unsigned char *pErrText )
{
	if( !(*pErrMk & ErrBit) ) {	/* Fehlerbit noch nicht gesetzt */
		*pErrMk |= ErrBit;
		ErrStatistics( pTaskName, ErrStat1, ErrNum, ErrInfo, pErrPre, pErrText );
	}
	else {
		ErrStatistics( pTaskName, ErrStatN, ErrNum, ErrInfo, pErrPre, pErrText );
	}
	if (pSyErr != NULL)
		*pSyErr += 1;
}

/*-----------------------------------------------------------------------------
// GetGlobalsPtr
// Liefert Zeiger auf Globaldatenstruktur
// Last Edit:
//		30.06.00/RES: ErrStatistics()-Aufruf bei Fehlern entfernt
//		19.07.99/RES
//		09.06.99/RES
//
// inputs:	-
// outputs: ppGlobals	Zeiger auf Globaldatenstruktur
// return:	-
//---------------------------------------------------------------------------*/
void GetGlobalsPtr( Globals_Typ **ppGlobals )
{
	static Globals_Typ *pGlobals = NULL;
	long lPtr, lVarLen;

	if( pGlobals == NULL ) {	/* Zeiger noch nicht bekannt ? */
		/* Zeiger auf Globaldatenstruktur ermitteln */
		if( !PV_xgetadr( "SYS_pGlobals", &lPtr, &lVarLen ) ) {
			pGlobals = *(Globals_Typ **)lPtr;
		}
		else {	/* SYS_pGlobals nicht gefunden */
			pGlobals = NULL;
		}
	}

	/* Zeiger zurueckliefern */
	*ppGlobals = pGlobals;
}
/*-----------------------------------------------------------------------------
// bin_to_bcd_8
// Wandelt Unsigned-long-Wert in 8-stellige BCD-Zahl (unsigned long) um
// Last Edit:
//		20.12.99/MKrz
//
// inputs:  value		Wert im Binaer-Format
//
// return:				Wert im BCD-Format
//---------------------------------------------------------------------------*/
unsigned long bin_to_bcd_8( unsigned long value )
{
	unsigned short	i;
	unsigned long	bcd = 0;
	unsigned long	tbin = 1;
	unsigned long	tbcd = 1;

	for (i=0; i<8; i++) {
		bcd += value/tbin % 10 * tbcd;
		tbin *= 10;
		tbcd *= 16;
	}
	return bcd;
}
```

#### bksysgetinfo.c
```c
#ifdef _DEFAULT_INCLUDES
	#include <AsDefault.h>
#endif
/* bksysgetinfo.c ------------------------------------------------------------- */

#include <bur/plc.h>      /*some usefull macros for B&R pcc programming*/

#include <stdlib.h>

#include "bksys.h"

/*-----------------------------------------------------------------------------
// GetDpInfo
// Sucht nach Datenpunkt mit angegebenem Namen und liefert interne Adresse und
// zugehoerigen Alias-Zeiger zurueck
// LastEdit:
//		22.02.02/RES	Rueckgabewert von GetDpInfo() geaendert (2=Leiche gefunden)
//		17.05.00/RES	PabSize von UCHAR auf USHORT geaendert (wg. BkZs)
//		22.09.99/RES	pPabHead und pDtDescr immer aktuell ermitteln
//		20.07.99/RES	Datenpunktname als Zeichenkette direkt im PAB
//		10.06.99/RES	Erstversion
//
// inputs:	pDpName		Datenpunktname (Zeichenkette)
// outputs:	pDtIdx		Datentyp-Index
//			pDpIdx		Datenpunkt-Index
//			ppAlias		Zeiger auf zugehoerige Alias-Struktur
// return:	 1 = Datenpunkt gefunden => Rueckgabe-Infos gueltig
//			 2 = Leiche gefunden => Rueckgabe-Infos gueltig
//			 0 = Keinen passenden Datenpunkt gefunden => Rueckgabe-Infos ungueltig
//			<0 = Bk2000-Systemfehler => Rueckgabe-Infos ungueltig
//---------------------------------------------------------------------------*/
short GetDpInfo( char *pDpName, unsigned char *pDtIdx, unsigned short *pDpIdx, unsigned char **ppAlias )
{
	short sFound = 0;
	unsigned char *pPab;
	unsigned char DtIdx;
	unsigned short DpIdx;
	unsigned short PabSize;
	unsigned char DpNameOff;
	Globals_Typ *pGlobals = NULL;
	PabHeader_Typ *pPabHead = NULL;
	DtProps_Typ *pDtProps = NULL;

	/* Zeiger auf Globaldatenstruktur initialisieren */
	GetGlobalsPtr( &pGlobals );
	if( pGlobals != NULL ) {	/* Gueltige Adresse in pGlobals ? */
		pPabHead = pGlobals->pPab;
		if( pPabHead == NULL ) {	/* Keine gueltige Adresse in pPab ? */
			return( -2 );
		}
		pDtProps = pGlobals->pDtProps;
		if( pDtProps == NULL ) {	/* Keine gueltige Adresse in pPab ? */
			return( -3 );
		}
	}
	else {	/* Keine gueltige Adresse in pGlobals */
		return( -1 );
	}

	/* Datenpunkt mittels Namen suchen */
	for( DtIdx = 0; !sFound && DtIdx < DT_ANZ; DtIdx++ ) {
		pPab = pPabHead->pDtBase[DtIdx];
		PabSize = pDtProps[DtIdx].DtPabLen;
		DpNameOff = pDtProps[DtIdx].DpNameOff;
		for( DpIdx = 0; DpIdx < pPabHead->DpAnz[DtIdx]; DpIdx++, pPab += PabSize ) {
			if( strcmp( pDpName, (char *)(pPab + DpNameOff) ) == 0 ) {
				*pDtIdx = *( pPab + pDtProps[DtIdx].DtIdxOff );
				*pDpIdx = *(unsigned short *)( pPab + pDtProps[DtIdx].DpIdxOff );
				*ppAlias = *(unsigned char **)( pPab + pDtProps[DtIdx].AliasPtrOff );
				if( *ppAlias != NULL ) {
					sFound = 1;	/* Datenpunkt mit passendem Namen gefunden */
				}
				else {
					sFound = 2;	/* Leiche im PAB gefunden */
				}
				break;
			}
		}
	}
	return( sFound );
}

/*-----------------------------------------------------------------------------
// GetDtDescInfos
// Liefert Zeiger und maximalen Eintragsindex von Datentyp-Deskriptoren und
// Item-Konvertierungtabellen
// Last Edit:
//		09.06.99/RES
//		06.06.99/RES
//
// inputs:	DtIdx			Datentyp-Index
// outputs: ppDtProps		Zeiger auf Datentyp-Eigenschaften
//			ppEaDesc		Zeiger auf Elementart-Descriptor
//			pEaDescMaxIdx	Hoechster Index in Elementart-Descriptor
//			ppDtDesc		Zeiger auf Datentyp-Descriptor
//			pDtDescMaxIdx	Hoechster Index in Datentyp-Descriptor
//			ppItemConv		Zeiger auf Item-Konvertierungstabelle
//			pItemConvMaxIdx	Hoechster Index in Item-Konvertierungstabelle
// return:	 0 = Rueckgabe-Infos gueltig
//			<0 = Fehler => Rueckgabe-Infos ungueltig
//---------------------------------------------------------------------------*/
short GetDtDescInfos( unsigned char DtIdx, DtProps_Typ **ppDtProps,
					  EaDesc_Typ **ppEaDesc, unsigned char *pEaDescMaxIdx,
					  DtDesc_Typ **ppDtDesc, unsigned char *pDtDescMaxIdx,
					  ItemConv_Typ **ppItemConv, unsigned char *pItemConvMaxIdx )
{
	static Globals_Typ *pGlobals = NULL;

	short sRet = 0;

	/* Zeiger auf Struktur mit Zeigern auf Globaldaten initialisieren */
	if( pGlobals == NULL ) {
		GetGlobalsPtr( &pGlobals );
	}

	if( pGlobals != NULL ) {
		/* Output-Informationen ermitteln */
		if( DtIdx < DT_ANZ ) {	/* Gueltiger Datentyp ? */
			/* Zeiger auf Struktur mit Datentyp-Eigenschaften */
			if( ppDtProps != NULL ) {
				*ppDtProps = pGlobals->pDtProps + DtIdx;
			}
			/* Zeiger auf Elementart-Deskriptor und zugehoerigen MaxIndex ermitteln */
			if( ppEaDesc != NULL ) {
				*ppEaDesc = pGlobals->pEaDesc[DtIdx];
			}
			if( pEaDescMaxIdx != NULL ) {
				*pEaDescMaxIdx = pGlobals->pDtProps[DtIdx].EaMaxItemIdx;
			}
			/* Zeiger auf Datentyp-Deskriptor und zugehoerigen MaxIndex ermitteln */
			if( ppDtDesc != NULL ) {
				*ppDtDesc = pGlobals->pDtDesc[DtIdx];
			}
			if( pDtDescMaxIdx != NULL ) {
				*pDtDescMaxIdx = pGlobals->pDtProps[DtIdx].DtMaxItemIdx;
			}
			/* Zeiger auf Itemkonvertierungstabelle und zugehoerigen MaxIndex ermitteln */
			if( ppItemConv != NULL ) {
				*ppItemConv = pGlobals->pItemConv[DtIdx];
			}
			if( pItemConvMaxIdx != NULL ) {
				*pItemConvMaxIdx = pGlobals->pDtProps[DtIdx].ItemConvMaxIdx;
			}
		}
		else {	/* Datentyp ungueltig */
			sRet = -1;
		}
	}
	else {	/* pGlobals == NULL */
		sRet = -2;
	}
	return( sRet );
}
```
